(* Schneider Machine Expert - Basic project CTF_OT_Challenge_2, file version 2.9.0.0 *)
(* ProjectInformations: Name=Nouveau projet *)

HARDWARE
  Cpu 0: TM221CE16T
  EthernetConfiguration: NetworkName=M221, IpAllocationMode=FixedAddress, IpAddress=192.168.1.4, SubnetMask=255.255.255.0
  SerialLineConfiguration: Baud=Baud19200, Parity=ParityEven, DataBits=DataBits8, StopBits=StopBits1, PhysicalMedium=PhysicalMediumRs485, TransmissionMode=TransmissionModeModbusRtu, SlaveId=1, Addressing=SlaveAddressing
  MastTask: UsePeriodScanMode=false, PeriodScan=100
  FastTask: Period=255
  CpuBehavior: StartingMode=StartInRun, AutoSaveRamOnEeprom=true, WatchdogPeriod=250

SYMBOLS  (address, symbol, comment, settings)
  %M11      AUTOPILOT
  %M13      CAPTAIN_CONTROL
  %M17      READY
  %M19      BALL_SENSOR
  %M23      POWDER_SENSOR
  %M29      GUN_UP
  %M31      LOAD_LOCKED
  %M37      FIRE_BLOCKED
  %M41      LOADER
  %M43      FIRE
  %M47      STOP_FIRE
  %M53      STOP_LOAD
  %M59      FORCE_FIRE
  %M61      FORCE_LOAD
  %M67      RAISE_GUN
  %M71      ARM
  %M83      CAPTAIN_TAKES_WHEEL
  %M123     BALL_READY_CMD
  %M177     POWDER_READY_CMD
  %M755     BALL_BLOCK
  %I0.0     START_MOTEUR  "Button start"
  %I0.1     STOP_MOTEUR  "Button stop"
  %Q0.0     MOTEUR  "Sortie commande moteur"

POU Nouveau POU
  (* SectionNumber=1 *)

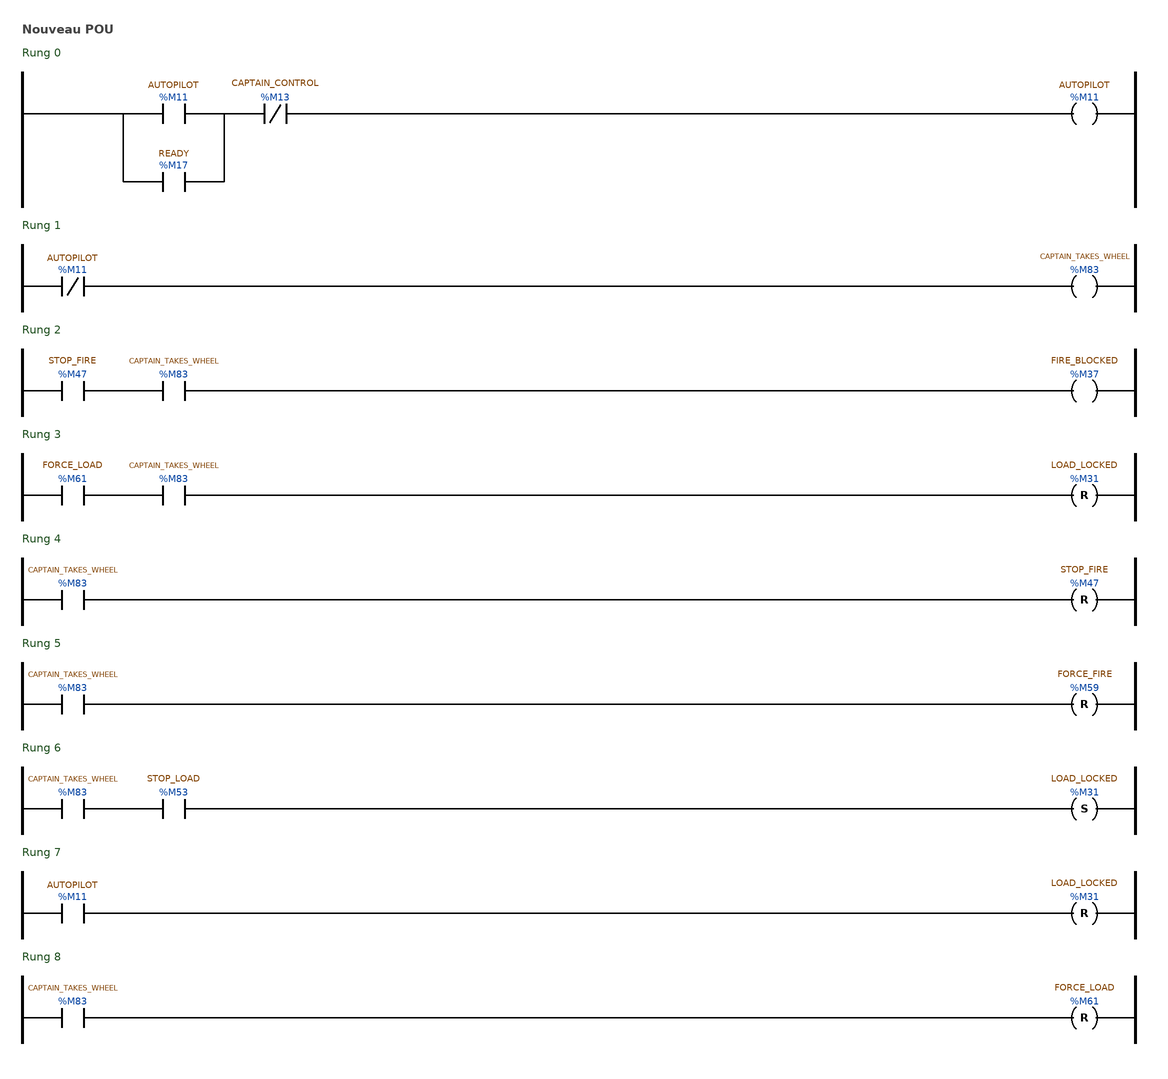

// Rung 0
  LD 1
  AND( %M11               (* AUTOPILOT *)
  OR %M17                 (* READY *)
  )
  ANDN %M13               (* CAPTAIN_CONTROL *)
  ST %M11                 (* AUTOPILOT *)
  // as ST:
  //   AUTOPILOT := (AUTOPILOT OR READY) AND NOT CAPTAIN_CONTROL;

// Rung 1
  LDN %M11                (* AUTOPILOT *)
  ST %M83                 (* CAPTAIN_TAKES_WHEEL *)
  // as ST:
  //   CAPTAIN_TAKES_WHEEL := NOT AUTOPILOT;

// Rung 2
  LD %M47                 (* STOP_FIRE *)
  AND %M83                (* CAPTAIN_TAKES_WHEEL *)
  ST %M37                 (* FIRE_BLOCKED *)
  // as ST:
  //   FIRE_BLOCKED := STOP_FIRE AND CAPTAIN_TAKES_WHEEL;

// Rung 3
  LD %M61                 (* FORCE_LOAD *)
  AND %M83                (* CAPTAIN_TAKES_WHEEL *)
  R %M31                  (* LOAD_LOCKED *)
  // as ST:
  //   IF FORCE_LOAD AND CAPTAIN_TAKES_WHEEL THEN LOAD_LOCKED := FALSE; END_IF;

// Rung 4
  LD %M83                 (* CAPTAIN_TAKES_WHEEL *)
  R %M47                  (* STOP_FIRE *)
  // as ST:
  //   IF CAPTAIN_TAKES_WHEEL THEN STOP_FIRE := FALSE; END_IF;

// Rung 5
  LD %M83                 (* CAPTAIN_TAKES_WHEEL *)
  R %M59                  (* FORCE_FIRE *)
  // as ST:
  //   IF CAPTAIN_TAKES_WHEEL THEN FORCE_FIRE := FALSE; END_IF;

// Rung 6
  LD %M83                 (* CAPTAIN_TAKES_WHEEL *)
  AND %M53                (* STOP_LOAD *)
  S %M31                  (* LOAD_LOCKED *)
  // as ST:
  //   IF CAPTAIN_TAKES_WHEEL AND STOP_LOAD THEN LOAD_LOCKED := TRUE; END_IF;

// Rung 7
  LD %M11                 (* AUTOPILOT *)
  R %M31                  (* LOAD_LOCKED *)
  // as ST:
  //   IF AUTOPILOT THEN LOAD_LOCKED := FALSE; END_IF;

// Rung 8
  LD %M83                 (* CAPTAIN_TAKES_WHEEL *)
  R %M61                  (* FORCE_LOAD *)
  // as ST:
  //   IF CAPTAIN_TAKES_WHEEL THEN FORCE_LOAD := FALSE; END_IF;

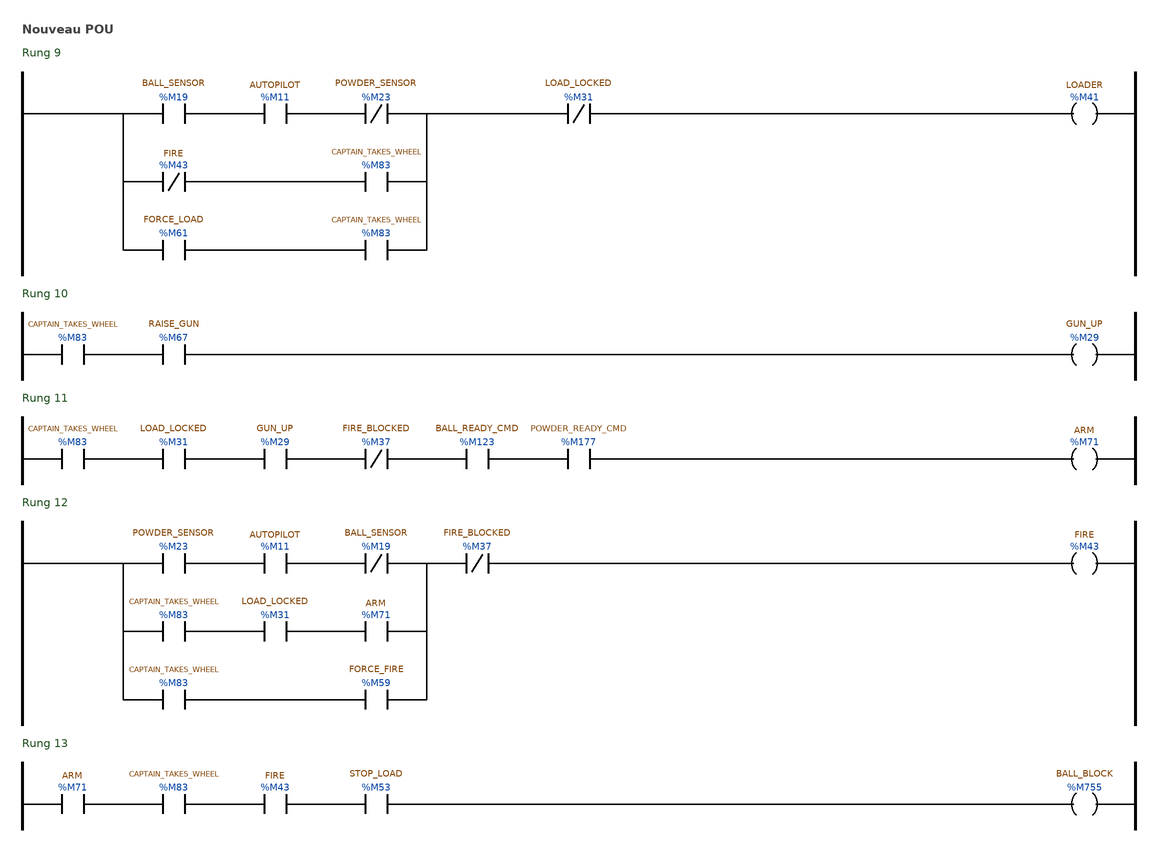

// Rung 9
  LD 1
  AND( %M19               (* BALL_SENSOR *)
  AND %M11                (* AUTOPILOT *)
  ANDN %M23               (* POWDER_SENSOR *)
  OR(N %M43               (* FIRE *)
  AND %M83                (* CAPTAIN_TAKES_WHEEL *)
  )
  OR( %M61                (* FORCE_LOAD *)
  AND %M83                (* CAPTAIN_TAKES_WHEEL *)
  )
  )
  ANDN %M31               (* LOAD_LOCKED *)
  ST %M41                 (* LOADER *)
  // as ST:
  //   LOADER := (BALL_SENSOR AND AUTOPILOT AND NOT POWDER_SENSOR OR NOT FIRE AND CAPTAIN_TAKES_WHEEL OR FORCE_LOAD AND CAPTAIN_TAKES_WHEEL) AND NOT LOAD_LOCKED;

// Rung 10
  LD %M83                 (* CAPTAIN_TAKES_WHEEL *)
  AND %M67                (* RAISE_GUN *)
  ST %M29                 (* GUN_UP *)
  // as ST:
  //   GUN_UP := CAPTAIN_TAKES_WHEEL AND RAISE_GUN;

// Rung 11
  LD %M83                 (* CAPTAIN_TAKES_WHEEL *)
  AND %M31                (* LOAD_LOCKED *)
  AND %M29                (* GUN_UP *)
  ANDN %M37               (* FIRE_BLOCKED *)
  AND %M123               (* BALL_READY_CMD *)
  AND %M177               (* POWDER_READY_CMD *)
  ST %M71                 (* ARM *)
  // as ST:
  //   ARM := CAPTAIN_TAKES_WHEEL AND LOAD_LOCKED AND GUN_UP AND NOT FIRE_BLOCKED AND BALL_READY_CMD AND POWDER_READY_CMD;

// Rung 12
  LD 1
  AND( %M23               (* POWDER_SENSOR *)
  AND %M11                (* AUTOPILOT *)
  ANDN %M19               (* BALL_SENSOR *)
  OR( %M83                (* CAPTAIN_TAKES_WHEEL *)
  AND %M31                (* LOAD_LOCKED *)
  AND %M71                (* ARM *)
  )
  OR( %M83                (* CAPTAIN_TAKES_WHEEL *)
  AND %M59                (* FORCE_FIRE *)
  )
  )
  ANDN %M37               (* FIRE_BLOCKED *)
  ST %M43                 (* FIRE *)
  // as ST:
  //   FIRE := (POWDER_SENSOR AND AUTOPILOT AND NOT BALL_SENSOR OR CAPTAIN_TAKES_WHEEL AND LOAD_LOCKED AND ARM OR CAPTAIN_TAKES_WHEEL AND FORCE_FIRE) AND NOT FIRE_BLOCKED;

// Rung 13
  LD %M71                 (* ARM *)
  AND %M83                (* CAPTAIN_TAKES_WHEEL *)
  AND %M43                (* FIRE *)
  AND %M53                (* STOP_LOAD *)
  ST %M755                (* BALL_BLOCK *)
  // as ST:
  //   BALL_BLOCK := ARM AND CAPTAIN_TAKES_WHEEL AND FIRE AND STOP_LOAD;

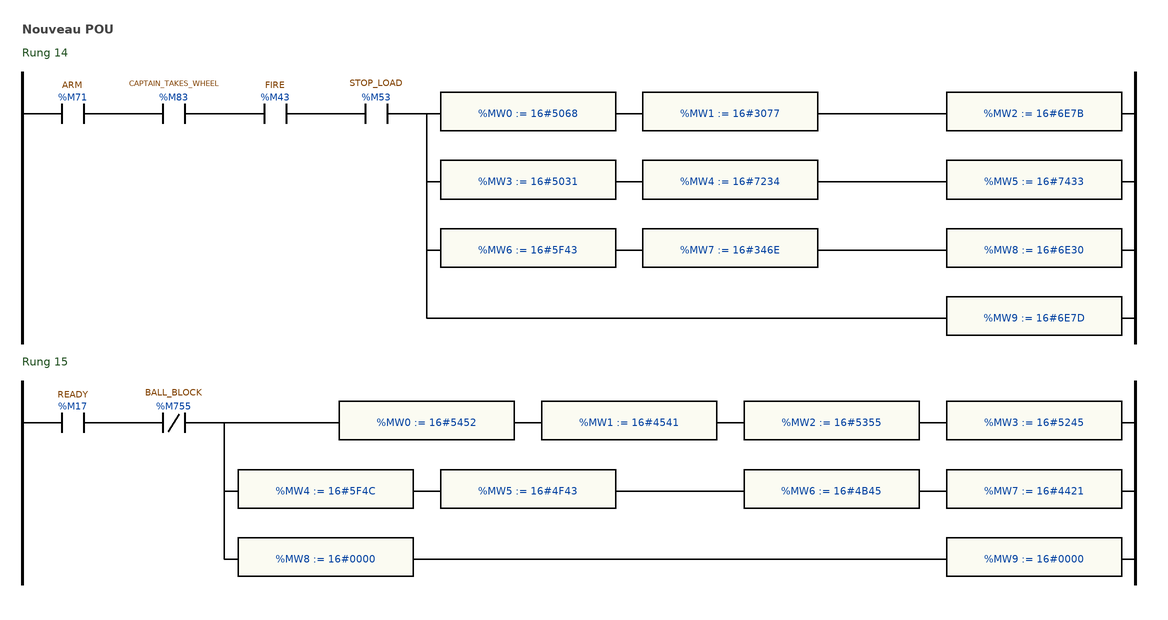

// Rung 14
  LD %M71                 (* ARM *)
  AND %M83                (* CAPTAIN_TAKES_WHEEL *)
  AND %M43                (* FIRE *)
  AND %M53                (* STOP_LOAD *)
  MPS
  OPER [ %MW0 := 16#5068 ]
  OPER [ %MW1 := 16#3077 ]
  [ %MW2 := 16#6E7B ]
  MRD
  OPER [ %MW3 := 16#5031 ]
  OPER [ %MW4 := 16#7234 ]
  [ %MW5 := 16#7433 ]
  MRD
  OPER [ %MW6 := 16#5F43 ]
  OPER [ %MW7 := 16#346E ]
  [ %MW8 := 16#6E30 ]
  MPP
  [ %MW9 := 16#6E7D ]
  // as ST:
  //   IF ARM AND CAPTAIN_TAKES_WHEEL AND FIRE AND STOP_LOAD THEN %MW0 := 16#5068; END_IF;
  //   IF ARM AND CAPTAIN_TAKES_WHEEL AND FIRE AND STOP_LOAD THEN %MW1 := 16#3077; END_IF;
  //   IF ARM AND CAPTAIN_TAKES_WHEEL AND FIRE AND STOP_LOAD THEN %MW2 := 16#6E7B; END_IF;
  //   IF ARM AND CAPTAIN_TAKES_WHEEL AND FIRE AND STOP_LOAD THEN %MW3 := 16#5031; END_IF;
  //   IF ARM AND CAPTAIN_TAKES_WHEEL AND FIRE AND STOP_LOAD THEN %MW4 := 16#7234; END_IF;
  //   IF ARM AND CAPTAIN_TAKES_WHEEL AND FIRE AND STOP_LOAD THEN %MW5 := 16#7433; END_IF;
  //   IF ARM AND CAPTAIN_TAKES_WHEEL AND FIRE AND STOP_LOAD THEN %MW6 := 16#5F43; END_IF;
  //   IF ARM AND CAPTAIN_TAKES_WHEEL AND FIRE AND STOP_LOAD THEN %MW7 := 16#346E; END_IF;
  //   IF ARM AND CAPTAIN_TAKES_WHEEL AND FIRE AND STOP_LOAD THEN %MW8 := 16#6E30; END_IF;
  //   IF ARM AND CAPTAIN_TAKES_WHEEL AND FIRE AND STOP_LOAD THEN %MW9 := 16#6E7D; END_IF;

// Rung 15
  LD %M17                 (* READY *)
  ANDN %M755              (* BALL_BLOCK *)
  MPS
  OPER [ %MW0 := 16#5452 ]
  OPER [ %MW1 := 16#4541 ]
  OPER [ %MW2 := 16#5355 ]
  [ %MW3 := 16#5245 ]
  MRD
  OPER [ %MW4 := 16#5F4C ]
  OPER [ %MW5 := 16#4F43 ]
  OPER [ %MW6 := 16#4B45 ]
  [ %MW7 := 16#4421 ]
  MPP
  OPER [ %MW8 := 16#0000 ]
  [ %MW9 := 16#0000 ]
  // as ST:
  //   IF READY AND NOT BALL_BLOCK THEN %MW0 := 16#5452; END_IF;
  //   IF READY AND NOT BALL_BLOCK THEN %MW1 := 16#4541; END_IF;
  //   IF READY AND NOT BALL_BLOCK THEN %MW2 := 16#5355; END_IF;
  //   IF READY AND NOT BALL_BLOCK THEN %MW3 := 16#5245; END_IF;
  //   IF READY AND NOT BALL_BLOCK THEN %MW4 := 16#5F4C; END_IF;
  //   IF READY AND NOT BALL_BLOCK THEN %MW5 := 16#4F43; END_IF;
  //   IF READY AND NOT BALL_BLOCK THEN %MW6 := 16#4B45; END_IF;
  //   IF READY AND NOT BALL_BLOCK THEN %MW7 := 16#4421; END_IF;
  //   IF READY AND NOT BALL_BLOCK THEN %MW8 := 16#0000; END_IF;
  //   IF READY AND NOT BALL_BLOCK THEN %MW9 := 16#0000; END_IF;
